// TIA Portal V15.1 export
// export: Created 2019-08-14T06:29:50.5674523Z, ExportSetting None, DisplayName Totally Integrated Automation Portal, DisplayVersion V15.1, DisplayName TIA Portal Openness, DisplayVersion V15.1, DisplayName STEP 7 Professional, DisplayVersion V15.1, DisplayName STEP 7 Safety, DisplayVersion V15.1, DisplayName WinCC Advanced, DisplayVersion V15.1
DATA_BLOCK "Skill_#SKILL_NAME#_DB"   // DB4
{ S7_Optimized_Access := 'TRUE' }
// stored: InstanceOfName Skill_#SKILL_NAME#, InstanceOfType FB
"Skill_#SKILL_NAME#"
   // VAR_INPUT
   //    ModulToSkill : "typeModulSkillInterface_IN";
   // END_VAR
   // VAR_OUTPUT
   //    SkillToModul : "typeModulSkillInterface_OUT";
   // END_VAR
   // VAR
   //    State { S7_SetPoint := 'True'} : UInt;
   //    StateOfExecute : UInt;
   //    ResultTrigger : DInt;
   //    ResultFeched : Bool;
   //    oldResultTrigger : DInt;
   //    NextStep : Bool;
   //    Parameter_In : "type#SKILL_NAME#StartParameter_In";
   //    Parameter_Out : "type#SKILL_NAME#GetResultParameter_Out";
   //    statErrorId { S7_SetPoint := 'True'} : Int;
   //    ResultAcknowledge : Bool;
   //    StartByMES { S7_SetPoint := 'True'} : Bool;
   //    rtStart : R_TRIG;
   //    rtStop : R_TRIG;
   //    rtAbort : R_TRIG;
   //    rtReset : R_TRIG;
   //    rtStep : R_TRIG;
   //    rtNextStep : R_TRIG;
   //    Start : "#SKILL_NAME#_Start";
   //    GetResult : "#SKILL_NAME#_GetResult";
   // END_VAR
BEGIN
END_DATA_BLOCK
